# EPICS substitutions: db/user.substitutions
# SPDX-FileCopyrightText: 2006 Argonne National Laboratory
#
# SPDX-License-Identifier: EPICS

# Example substitutions file

file "db/circle.db" {
    { user = "Administrator" }
}

file "db/dbExample1.db" {
    { user = "Administrator" }
}

file db/dbExample2.db {
    pattern { user, no, scan }
        { "Administrator", 1, "1 second" }
        { "Administrator", 2, "2 second" }
        { "Administrator", 3, "5 second" }
}
